TYPE tstCTCInternalCommands :
STRUCT
	bHome 			:BOOL;
	bTeach 			:BOOL;
	bMoveAbsolute 	:BOOL;
	bHalt 			:BOOL;
	bMoveIn 		:BOOL;
	bMoveOut 		:BOOL;
	bMoveContinuous :BOOL;
END_STRUCT
END_TYPE

(* stored: Version 1.1.0.1, ProductVersion 3.1.4026.17
   DUT tstCTCInternalCommands: Id {77c492d9-04dd-43d1-896b-9daa9c88b7ca} *)
